TYPE st_HMItoPLC_VariantControl :
STRUCT
    bExportJSON : BOOL;
    bWriteJSON : BOOL;
    Config : ST_Configuration;
    bNeedsCellDefinition : BOOL;
END_STRUCT
END_TYPE

(* stored: Version 1.1.0.1, ProductVersion 3.1.4024.9
   DUT st_HMItoPLC_VariantControl: Id {87811677-9a09-4767-bbea-e680f216aec1} *)
